TYPE ST_HW_OutputsProBoxElementMotor :
(**************************************************************************************
 * 	Application		:	BoxControl Framework
 *	Revision		:	$Revision: 417092 $
 *	Revision date	:	$Date: 2018-11-14 12:58:58 +0100 (Wed, 14 Nov 2018) $
 *	Last changed by	:	$Author: q8aberh $
 *	URL				:	$URL: http://almscdc.swisslog.com/repo/SWPD/Development/ProMove/02_Controls/ProBox/03_Implementation/01_DevelopmentProject/01_Software/ProBox_COE/ProBox_DevProj_v1.0/PLC_1/20_Product/10_App/13_Elements/10_Lib/11_ProBox/11_ElementMotor/01_DUTs/ST_HW_Outp $
 *
 *	Purpose			:	Dummy Element motor - Hardware outputs
 *
 * ------------------------------------------------------------------------------------
 *	Copyright Swisslog [IP AG], Switzerland. All rights reserved.
 * 
 * ------------------------------------------------------------------------------------
 *	
 * 	Revision History: 
 *
 * 	VERSION			DATE			INITIALS			DESCRIPTION
 *	0.1				13.04.2018		PkF					First version of outputs for a motor on a element
 *
 **************************************************************************************)
STRUCT
	Drive_Run_12 		: BOOL; // Drive run command axis 1-2 forward
	Drive_Run_21 		: BOOL; // Drive run command axis 1-2 reverse
	Drive_Creep_12 		: BOOL; // Drive creep speed command axis 1-2
	Drive_Low_12 		: BOOL; // Drive low speed command axis 1-2	
	MotorBrake_12		: BOOL; // Release brake axis 1-2
END_STRUCT
END_TYPE

(* stored: Version 1.1.0.1, ProductVersion 3.1.4022.12
   DUT ST_HW_OutputsProBoxElementMotor: Id {d0289788-745e-44ff-8e07-e38704713c90} *)
